// TIA Portal project "Project3" (V15)
// Vorlageprojekt für das Buch mit Zielsystem S7-1200

(* hardware
DEVICE "S7-1200-Station_1"  S7-1200 Station
   slot 0: "Baugruppenträger_0"  Rack  V1.0
   slot 1: "PLC_1"  CPU 1211C DC/DC/DC  6ES7 211-1AE40-0XB0  V4.1
*)

// ===== PLC "PLC_1"  CPU 1211C DC/DC/DC =====

VAR_GLOBAL   // PLC tag table "Standard-Variablentabelle"
   "START" AT %I0.0 : Bool;
   "STOP" AT %I0.1 : Bool;
   "SENSOR 1" AT %I0.2 : Bool;
   "SENSOR 2" AT %I0.4 : Bool;
   "SENSOR 3" AT %I0.5 : Bool;
   "BELT 6cm" AT %Q0.0 : Bool;
   "BELT 2m 1" AT %Q0.1 : Bool;
   "BELT 2m 2" AT %Q0.2 : Bool;
   "X" AT %M0.1 : Bool;
   "SENSOR 4" AT %I0.3 : Bool;
   "BELT 2m 3" AT %Q0.3 : Bool;
   "BELT 2m 4" AT %Q0.4 : Bool;
   "C BELT" AT %Q0.5 : Bool;
   "ARM 1" AT %Q0.6 : Bool;
   "BELT ARM 1" AT %Q0.7 : Bool;
   "ARM 2" AT %Q1.0 : Bool;
   "BELT ARM 2" AT %Q1.1 : Bool;
   "ARM 3" AT %Q1.2 : Bool;
   "BELT ARM 3" AT %Q1.3 : Bool;
   "Tag_1" AT %M0.2 : Bool;
   "Tag_2" AT %M0.3 : Bool;
   "Tag_3" AT %M1.0 : Bool;
   "Tag_4" AT %M1.1 : Bool;
   "Tag_5" AT %M1.2 : Bool;
   "Tag_6" AT %M1.3 : Bool;
END_VAR

FUNCTION "MHJ-PLC-Lab-Function-S71200" : Void   // FC9000, SCL
{ S7_Optimized_Access := 'TRUE' }
VERSION : 0.1
   VAR_TEMP
      rdTimeReturn : Int;
      outputTime : DTL;
      SyncVal : Byte;
      forVal : Int;
      forVal_2 : Int;
      Value : Byte;
   END_VAR
   VAR CONSTANT
      CompVal : Byte := 16#34;
      Value_01 : Byte := 16#11;
      Value_01_DW : DWord := 16#A165_D992;
      Value_02_DW : DWord := 16#58BE_4401;
   END_VAR
BEGIN

   #Value:=PEEK(area := 16#82,
        dbNumber := 0,
        byteOffset := 511);
   #Value := #Value + 1;

   POKE(area := 16#82,
        dbNumber := 0,
        byteOffset := 511,
        value := #Value);

   POKE(area:=16#81,
        dbNumber:=0,
        byteOffset:=1016,
        value:=#Value_01_DW);
   POKE(area := 16#81,
        dbNumber := 0,
        byteOffset := 1020,
        value := #Value_02_DW);

   POKE(area := 16#81,
        dbNumber := 0,
        byteOffset := 511,
        value := B#16#00);

   FOR #forVal := 0 TO 120 DO
       FOR #forVal_2:=0 TO 10 DO
           #rdTimeReturn:=RD_SYS_T(#outputTime);
           #rdTimeReturn := WR_SYS_T(#outputTime);
           #rdTimeReturn := RD_SYS_T(#outputTime);
           #rdTimeReturn := WR_SYS_T(#outputTime);
       END_FOR;
       #SyncVal:= PEEK(area := 16#81,
                      dbNumber := 0,
                      byteOffset := 511);
       IF #SyncVal = #CompVal THEN
          GOTO M_1;
       END_IF;
   END_FOR;
   RETURN;

   M_1:
   POKE(area := 16#81,
        dbNumber := 0,
        byteOffset := 511,
        value := B#16#0);
END_FUNCTION

ORGANIZATION_BLOCK "Main"   // OB1, LAD, ProgramCycle
TITLE = "Main Program Sweep (Cycle)"
{ S7_Optimized_Access := 'TRUE' }
VERSION : 0.1
   VAR_INPUT
      Initial_Call : Bool;   // Initial call of this OB
      Remanence : Bool;   // =True, if remanent data are available
   END_VAR
   VAR_TEMP   // added for the SCL form of the ladder/FBD networks
      _w1 : Bool;
      _w2 : Bool;
   END_VAR
BEGIN

REGION Network 1: Konnektierungsbaustein für PLC-Lab
   // Im Netzwerk 1 wird der Konnektierungsbaustein für PLC-Lab aufgerufen.
   // Dieser Aufruf darf nicht entfernt werden!
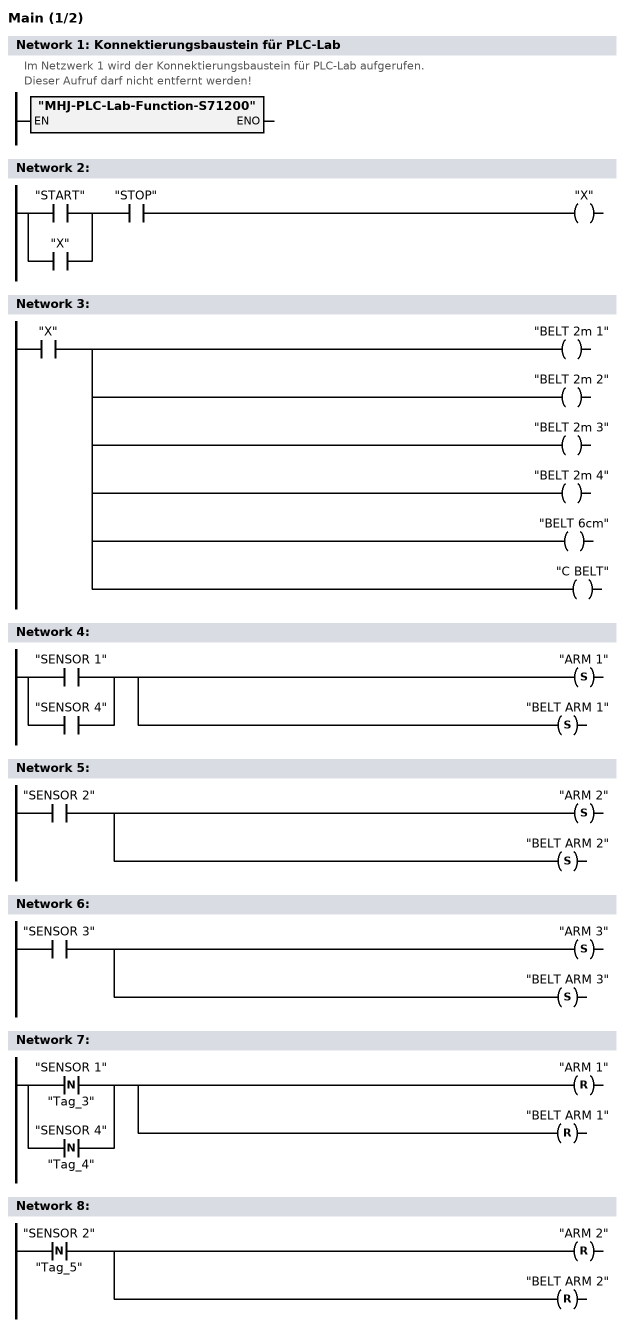
   RUNG wire#powerrail
      "MHJ-PLC-Lab-Function-S71200"()
   END_RUNG
   // the same network as SCL:
   "MHJ-PLC-Lab-Function-S71200"();
END_REGION

REGION Network 2
   RUNG wire#powerrail
      Contact( "START" )
      wire#w1
      Contact( "STOP" )
      Coil( "X" )
   END_RUNG
   RUNG wire#powerrail
      Contact( "X" )
   END_RUNG wire#w1
   // the same network as SCL:
   "X" := ("START" OR "X") AND "STOP";
END_REGION

REGION Network 3
   RUNG wire#powerrail
      Contact( "X" )
      wire#w1
      Coil( "BELT 2m 1" )
   END_RUNG
   RUNG wire#w1
      Coil( "BELT 2m 2" )
   END_RUNG
   RUNG wire#w1
      Coil( "BELT 2m 3" )
   END_RUNG
   RUNG wire#w1
      Coil( "BELT 2m 4" )
   END_RUNG
   RUNG wire#w1
      Coil( "BELT 6cm" )
   END_RUNG
   RUNG wire#w1
      Coil( "C BELT" )
   END_RUNG
   // the same network as SCL:
   "BELT 2m 1" := "X";
   "BELT 2m 2" := "X";
   "BELT 2m 3" := "X";
   "BELT 2m 4" := "X";
   "BELT 6cm" := "X";
   "C BELT" := "X";
END_REGION

REGION Network 4
   RUNG wire#powerrail
      Contact( "SENSOR 1" )
      wire#w1
      S_Coil( "ARM 1" )
   END_RUNG
   RUNG wire#powerrail
      Contact( "SENSOR 4" )
   END_RUNG wire#w1
   RUNG wire#w1
      S_Coil( "BELT ARM 1" )
   END_RUNG
   // the same network as SCL:
   IF "SENSOR 1" OR "SENSOR 4" THEN
       "ARM 1" := TRUE;
       "BELT ARM 1" := TRUE;
   END_IF;
END_REGION

REGION Network 5
   RUNG wire#powerrail
      Contact( "SENSOR 2" )
      wire#w1
      S_Coil( "ARM 2" )
   END_RUNG
   RUNG wire#w1
      S_Coil( "BELT ARM 2" )
   END_RUNG
   // the same network as SCL:
   IF "SENSOR 2" THEN
       "ARM 2" := TRUE;
       "BELT ARM 2" := TRUE;
   END_IF;
END_REGION

REGION Network 6
   RUNG wire#powerrail
      Contact( "SENSOR 3" )
      wire#w1
      S_Coil( "ARM 3" )
   END_RUNG
   RUNG wire#w1
      S_Coil( "BELT ARM 3" )
   END_RUNG
   // the same network as SCL:
   IF "SENSOR 3" THEN
       "ARM 3" := TRUE;
       "BELT ARM 3" := TRUE;
   END_IF;
END_REGION

REGION Network 7
   RUNG wire#powerrail
      N_Contact(operand := "SENSOR 1", bit := "Tag_3")
      wire#w1
      R_Coil( "ARM 1" )
   END_RUNG
   RUNG wire#powerrail
      N_Contact(operand := "SENSOR 4", bit := "Tag_4")
   END_RUNG wire#w1
   RUNG wire#w1
      R_Coil( "BELT ARM 1" )
   END_RUNG
   // the same network as SCL:
   #_w1 := NOT "SENSOR 1" AND "Tag_3";   // falling edge of "SENSOR 1"
   "Tag_3" := "SENSOR 1";
   #_w2 := NOT "SENSOR 4" AND "Tag_4";   // falling edge of "SENSOR 4"
   "Tag_4" := "SENSOR 4";
   IF #_w1 OR #_w2 THEN
       "ARM 1" := FALSE;
       "BELT ARM 1" := FALSE;
   END_IF;
END_REGION

REGION Network 8
   RUNG wire#powerrail
      N_Contact(operand := "SENSOR 2", bit := "Tag_5")
      wire#w1
      R_Coil( "ARM 2" )
   END_RUNG
   RUNG wire#w1
      R_Coil( "BELT ARM 2" )
   END_RUNG
   // the same network as SCL:
   #_w1 := NOT "SENSOR 2" AND "Tag_5";   // falling edge of "SENSOR 2"
   "Tag_5" := "SENSOR 2";
   IF #_w1 THEN
       "ARM 2" := FALSE;
       "BELT ARM 2" := FALSE;
   END_IF;
END_REGION

REGION Network 9
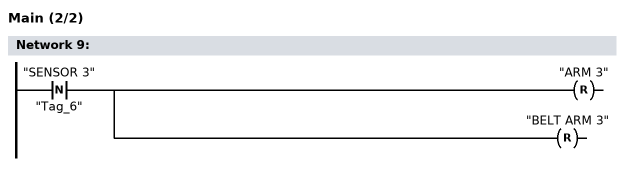
   RUNG wire#powerrail
      N_Contact(operand := "SENSOR 3", bit := "Tag_6")
      wire#w1
      R_Coil( "ARM 3" )
   END_RUNG
   RUNG wire#w1
      R_Coil( "BELT ARM 3" )
   END_RUNG
   // the same network as SCL:
   #_w1 := NOT "SENSOR 3" AND "Tag_6";   // falling edge of "SENSOR 3"
   "Tag_6" := "SENSOR 3";
   IF #_w1 THEN
       "ARM 3" := FALSE;
       "BELT ARM 3" := FALSE;
   END_IF;
END_REGION
END_ORGANIZATION_BLOCK